{attribute 'GeneratedUsingTerminal: EP6224-2022-0016'}
{attribute addProperty BoxType "EP6224-2022-0016"}
{attribute addProperty Id "EMPTY_STRUCTURE"}
{attribute addProperty CRC "0"}
{attribute addProperty Size "0"}
TYPE EMPTY_STRUCTURE :
STRUCT
END_STRUCT
END_TYPE

(* stored: Version 1.2.0.0, ProductVersion 3.1.4024.9
   DUT EMPTY_STRUCTURE: Id {92902f4e-5ec1-4598-829e-567bd9ce6c4b} *)
